FUNCTION_BLOCK FB_SimCapper
VAR_INPUT
END_VAR
VAR_OUTPUT
END_VAR
VAR
	bClamp						AT %I* : BOOL;
	bCapTrigger					AT %I* : BOOL;
	bCapDone					AT %Q* : BOOL;
	bCapFail					AT %Q* : BOOL;
	bPartPresent				AT %Q* : BOOL;
	
	rand						: DRAND;
	iCapMs						: DINT;
	tmrCap						: TON;
	iState						: DINT;
END_VAR
VAR CONSTANT
	CHANCE_FAIL					: LREAL := 0.01;
END_VAR

rand(Seed:=117);

CASE iState OF
	0:
		IF bCapTrigger THEN
			iState := 10;
			iCapMs := 1000 + TO_DINT(rand.Num * 100);
		ELSE
			bCapDone := FALSE;
			bCapFail := FALSE;
		END_IF
		
	10:
		tmrCap(IN:=TRUE, PT:=TO_TIME(iCapMs));
		IF tmrCap.Q THEN
			tmrCap(IN:=FALSE);
			IF rand.Num < CHANCE_FAIL THEN
				bCapFail := TRUE;
			END_IF
			bCapDone := TRUE;
			iState := 20;
		END_IF
		
	20:
		iState := 0;
		
END_CASE

END_FUNCTION_BLOCK

(* stored: Version 1.1.0.1, ProductVersion 3.1.4024.12
   POU FB_SimCapper: Id {3ab80ab6-5b4a-46b9-ad1a-33a3418ccbd2}, SpecialFunc None *)
